PROGRAM MAIN
VAR
END_VAR

END_PROGRAM

(* stored: Version 1.1.0.1
   POU MAIN: Id {e4a61645-5778-4dce-95bd-2b96fec842c8} *)
